// SIMATIC S7-200 project (STEP 7-Micro/WIN), CPU 224XP REL 02.01

SYMBOL_TABLE Símbolos S7-200
Siempre_ON       SM0.0    // Siempre ON
END_SYMBOL_TABLE

ORGANIZATION_BLOCK PRINCIPAL:OB1
TITLE=COMENTARIOS DEL PROGRAMA
BEGIN
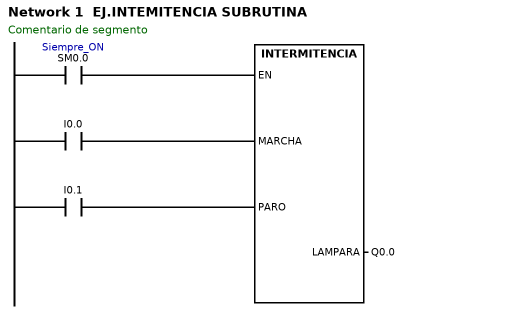
Network 1 // EJ.INTEMITENCIA SUBRUTINA
// Comentario de segmento
LD     Siempre_ON:SM0.0
=      L60.0
LD     I0.0
=      L63.7
LD     I0.1
=      L63.6
LD     L60.0
CALL   INTERMITENCIA:SBR0, L63.7, L63.6, Q0.0
END_ORGANIZATION_BLOCK

SUBROUTINE_BLOCK INTERMITENCIA:SBR0
TITLE=COMENTARIOS DE LA SUBRUTINA
VAR_INPUT
MARCHA:BOOL;	// L0.0 
PARO:BOOL;	// L0.1 
END_VAR
VAR_OUTPUT
LAMPARA:BOOL;	// L0.2 
END_VAR
VAR
AUXILIAR:BOOL;	// L0.3 
END_VAR
BEGIN
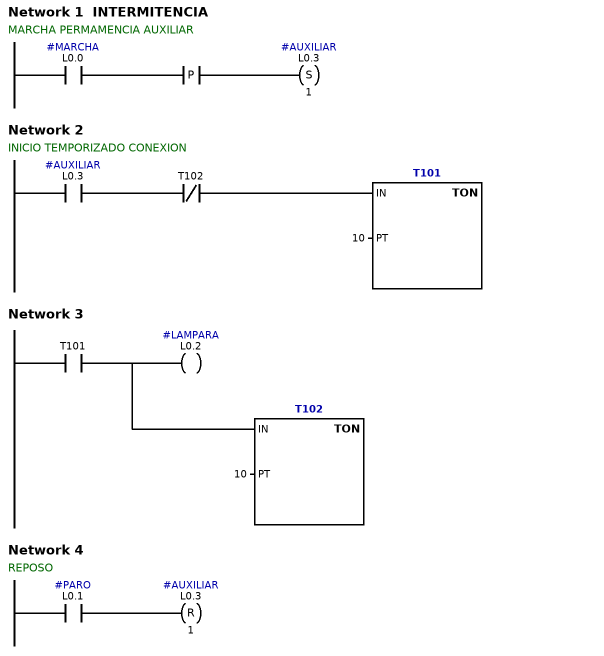
Network 1 // INTERMITENCIA
// MARCHA PERMAMENCIA AUXILIAR
LD     #MARCHA:L0.0
EU
S      #AUXILIAR:L0.3, 1
Network 2
// INICIO TEMPORIZADO CONEXION
LD     #AUXILIAR:L0.3
AN     T102
TON    T101, 10
Network 3
LD     T101
=      #LAMPARA:L0.2
TON    T102, 10
Network 4
// REPOSO
LD     #PARO:L0.1
R      #AUXILIAR:L0.3, 1
END_SUBROUTINE_BLOCK
